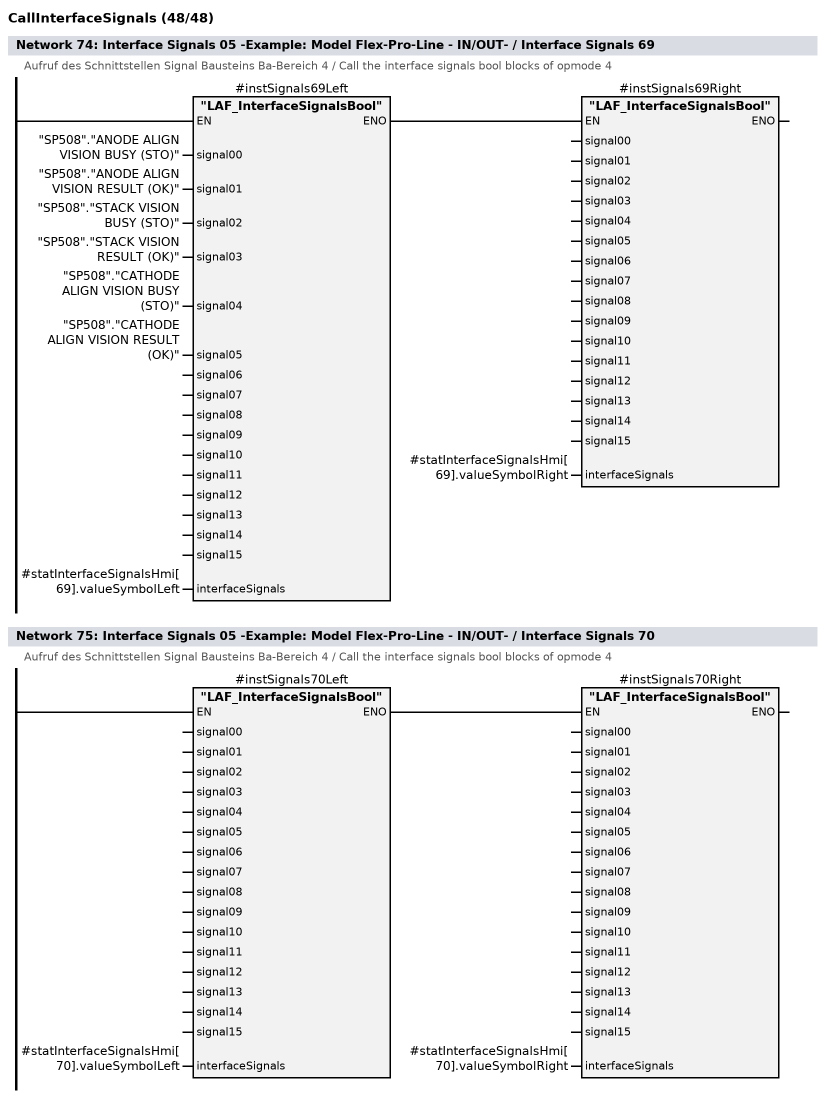
   RUNG wire#powerrail
      #instSignals69Left(signal00 := "SP508"."ANODE ALIGN VISION BUSY (STO)", signal01 := "SP508"."ANODE ALIGN VISION RESULT (OK)", signal02 := "SP508"."STACK VISION BUSY (STO)", signal03 := "SP508"."STACK VISION RESULT (OK)", signal04 := "SP508"."CATHODE ALIGN VISION BUSY (STO)", signal05 := "SP508"."CATHODE ALIGN VISION RESULT (OK)", signal06 :=, signal07 :=, signal08 :=, signal09 :=, signal10 :=, signal11 :=, signal12 :=, signal13 :=, signal14 :=, signal15 :=, interfaceSignals := #statInterfaceSignalsHmi[69].valueSymbolLeft)
      #instSignals69Right(signal00 :=, signal01 :=, signal02 :=, signal03 :=, signal04 :=, signal05 :=, signal06 :=, signal07 :=, signal08 :=, signal09 :=, signal10 :=, signal11 :=, signal12 :=, signal13 :=, signal14 :=, signal15 :=, interfaceSignals := #statInterfaceSignalsHmi[69].valueSymbolRight)
   END_RUNG
   // the same network as SCL:
   #instSignals69Left(signal00 := "SP508"."ANODE ALIGN VISION BUSY (STO)",   // "LAF_InterfaceSignalsBool"
                      signal01 := "SP508"."ANODE ALIGN VISION RESULT (OK)",
                      signal02 := "SP508"."STACK VISION BUSY (STO)",
                      signal03 := "SP508"."STACK VISION RESULT (OK)",
                      signal04 := "SP508"."CATHODE ALIGN VISION BUSY (STO)",
                      signal05 := "SP508"."CATHODE ALIGN VISION RESULT (OK)",
                      interfaceSignals := #statInterfaceSignalsHmi[69].valueSymbolLeft,
                      ENO => #_w1);
   IF #_w1 THEN
       #instSignals69Right(interfaceSignals := #statInterfaceSignalsHmi[69].valueSymbolRight);   // "LAF_InterfaceSignalsBool"
   END_IF;
END_REGION

REGION Network 75: Interface Signals 05 -Example: Model Flex-Pro-Line - IN/OUT- / Interface Signals 70
   // Aufruf des Schnittstellen Signal Bausteins Ba-Bereich 4 / Call the interface signals bool blocks of opmode 4
   RUNG wire#powerrail
      #instSignals70Left(signal00 :=, signal01 :=, signal02 :=, signal03 :=, signal04 :=, signal05 :=, signal06 :=, signal07 :=, signal08 :=, signal09 :=, signal10 :=, signal11 :=, signal12 :=, signal13 :=, signal14 :=, signal15 :=, interfaceSignals := #statInterfaceSignalsHmi[70].valueSymbolLeft)
      #instSignals70Right(signal00 :=, signal01 :=, signal02 :=, signal03 :=, signal04 :=, signal05 :=, signal06 :=, signal07 :=, signal08 :=, signal09 :=, signal10 :=, signal11 :=, signal12 :=, signal13 :=, signal14 :=, signal15 :=, interfaceSignals := #statInterfaceSignalsHmi[70].valueSymbolRight)
   END_RUNG
   // the same network as SCL:
   #instSignals70Left(interfaceSignals := #statInterfaceSignalsHmi[70].valueSymbolLeft, ENO => #_w1);   // "LAF_InterfaceSignalsBool"
   IF #_w1 THEN
       #instSignals70Right(interfaceSignals := #statInterfaceSignalsHmi[70].valueSymbolRight);   // "LAF_InterfaceSignalsBool"
   END_IF;
END_REGION
END_FUNCTION_BLOCK
